// LS Electric XG5000 project: Master
// PLC LSPLC

PROGRAM NewProgram (task: Scan Program)

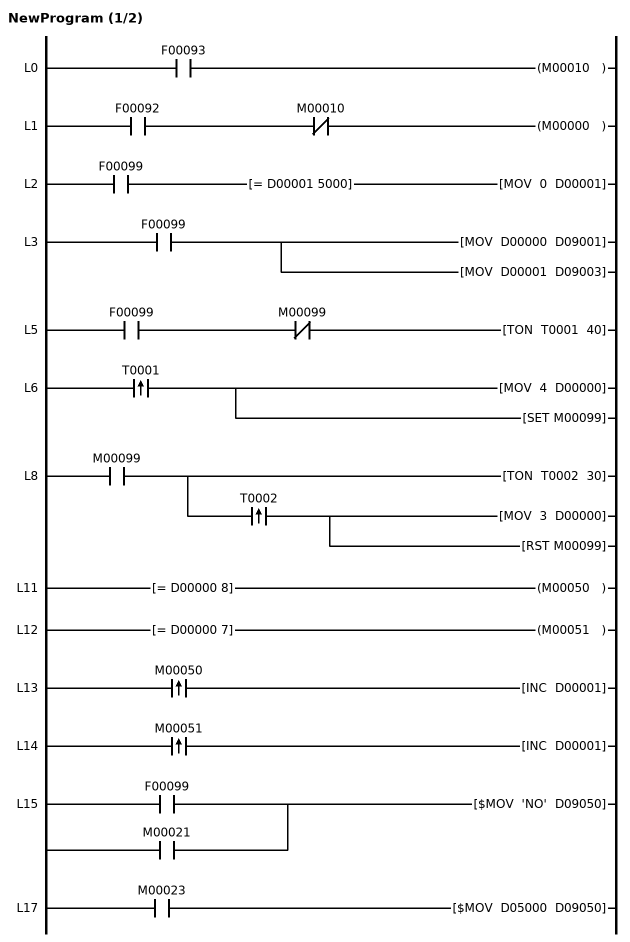
; L0
LOAD      F00093
OUT       M00010
; L1
LOAD      F00092
AND NOT   M00010
OUT       M00000
; L2
LOAD      F00099
AND=      D00001 5000
MOV       0 D00001
; L3
LOAD      F00099
MOV       D00000 D09001
MOV       D00001 D09003
; L5
LOAD      F00099
AND NOT   M00099
TON       T0001 40
; L6
LOADP     T0001
MOV       4 D00000
SET       M00099
; L8
LOAD      M00099
TON       T0002 30
ANDP      T0002
MOV       3 D00000
RST       M00099
; L11
LOAD=     D00000 8
OUT       M00050
; L12
LOAD=     D00000 7
OUT       M00051
; L13
LOADP     M00050
INC       D00001
; L14
LOADP     M00051
INC       D00001
; L15
LOAD      F00099
OR        M00021
$MOV      'NO' D09050
; L17
LOAD      M00023
$MOV      D05000 D09050

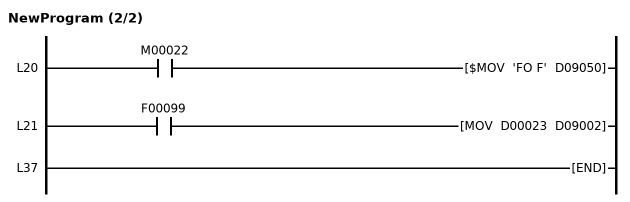
; L20
LOAD      M00022
$MOV      'FO F' D09050
; L21
LOAD      F00099
MOV       D00023 D09002
; L37
END